Staubli VAL3: RemoteAxisCtrl.pjx

--- RemoteAxisCtrl.pjx ---
Parameters version=s7.3.1 stackSize=5000 millimeterUnit=true
Program file=Comunicacion.pgx
Program file=JOGG_PC.pgx
Program file=init.pgx
Program file=set_sign.pgx
Program file=start.pgx
Program file=stop.pgx
Data file=RemoteAxisCtrl.dtx

--- RemoteAxisCtrl.dtx ---
bool bABSOLUTE = true
bool bBLOQ_CTRL
bool bBusy
bool bError
bool bHoming = true
bool bNewMove
bool bSTOP = true
bool bSync = true
dio Electrovalvule[2]
  [0] = {link=valve1}
  [1] = {link=valve2}
dio dBIO_salidas[4]
  [0] = {link=BasicIO-1\%Q0}
  [1] = {link=BasicIO-1\%Q1}
  [2] = {link=BasicIO-1\%Q2}
  [3] = {link=BasicIO-1\%Q3}
jointRx home = {j2=60, j3=60, j5=60}
jointRx jActualPos = {j2=60, j3=60, j5=60}
jointRx jError = {j1=0.1, j2=0.1, j3=0.1, j4=0.1, j5=0.1, j6=0.1}
jointRx jdestino = {j2=60, j3=60, j5=60}
jointRx origen
mdesc mNomSpeed = {blend=off}
mdesc mSpeed = {vel=10, blend=off}
num action
num axis_v[6]
  [5] = 1
num d_min = 0.5
num error_code
num g_data[82]
  [0] = 156
  [1] = 124
  [2] = 66
  [3] = 89
  [4] = 39
  [5] = 121
  [6] = 244
  [7] = 77
  [12] = 66
  [18] = 128
  [20] = 20
  [21] = 10
  [42] = 100
num g_message_send[82]
  [0] = 156
  [1] = 124
  [2] = 66
  [3] = 89
  [4] = 39
  [5] = 121
  [6] = 244
  [7] = 77
  [12] = 66
  [16] = 32
  [20] = 20
  [21] = 10
  [22] = 250
  [23] = 202
  [26] = 208
  [27] = 7
  [30] = 64
  [31] = 31
  [34] = 80
  [35] = 70
  [42] = 80
  [43] = 70
  [48] = 1
  [49] = 1
  [51] = 1
num id = -1
num id_actual = -2
num joint_v[6]
num mode_mov
num move_inc = 1
num nBytes
num n_status = 1
num speed = 10
num working_mode
pointRx pActualPos = {x=519.615242, y=20, z=-80, rx=-180, rz=-180, shoulder=lefty, elbow=epositive, wrist=wpositive, fatherId=world[0]}
pointRx pPunto = {fatherId=world[0]}
pointRx pdestino = {x=539.615242, y=40, z=-60, rx=-160, ry=20, rz=-160, shoulder=lefty, elbow=epositive, wrist=wpositive, fatherId=world[0]}
sio sSockPC = {link=Socket\RemoteCTRL}
tool tGripper = {fatherId=flange[0], ioLink=valve1}

--- start.pgx ---
program start()
begin
  call init()

  while (bBLOQ_CTRL==false)
    call Comunicacion()
    call JOGG_PC()
    delay(0)
  endWhile

end

--- Comunicacion.pgx ---
program Comunicacion()
  local num i
  local num aux
begin
  //while salir==false
  //communication with the PC
  //Waiting a message from the PC
  nBytes=sioGet(sSockPC,g_data)
  if (nBytes>0)
    //A message was received
    //Reading Identification message (8 bytes). It'll be used in the answer.
    for i=0 to 7
      g_message_send[i]=g_data[i]
    endFor
    //Reserved bytes 8, 9, 10, 11
    //ACTION BYTE 12
    action=g_data[12]
    g_message_send[12]=action
    //Bytes 13, 14 (input reserved). Output -> Status*********************
    //Byte 15 (output error code)******************************
    switch (action)
      case 13
        //NULL ACTION
        //do not do anything.
      break
      case 16
        //READ DATA
        //Update the return data
        //ID message already done
        //Reserved 8, 9, 10, 11
        //ACTION done
        //Status
        g_message_send[13]=n_status
        g_message_send[14]=0
        //Error code
        g_message_send[15]=error_code
        //working mode
        g_message_send[16]=working_mode
        //electrovalvule
        g_message_send[17]=dioGet(Electrovalvule)
        //digital output
        g_message_send[18]=dioGet(dBIO_salidas)
        //DO reserved
        g_message_send[19]=0
        //move inc
        g_message_send[20]=move_inc
        //speed
        g_message_send[21]=speed
        //Actual pos axis
        pActualPos=here(tGripper,world)
        jActualPos=herej()
        call set_sign()
        if (mode_mov==1 or mode_mov==2)
          pActualPos=here(tGripper,world)
          for i=0 to 3
            g_message_send[22+i]=(bAnd(round(abs(pActualPos.trsf.x)*100),power(2,8*(i+1))-power(2,8*i)))/(power(2,8*i))
            g_message_send[26+i]=(bAnd(round(abs(pActualPos.trsf.y)*100),power(2,8*(i+1))-power(2,8*i)))/(power(2,8*i))
            g_message_send[30+i]=(bAnd(round(abs(pActualPos.trsf.z)*100),power(2,8*(i+1))-power(2,8*i)))/(power(2,8*i))
            g_message_send[34+i]=(bAnd(round(abs(pActualPos.trsf.rx)*100),power(2,8*(i+1))-power(2,8*i)))/(power(2,8*i))
            g_message_send[38+i]=(bAnd(round(abs(pActualPos.trsf.ry)*100),power(2,8*(i+1))-power(2,8*i)))/(power(2,8*i))
            g_message_send[42+i]=(bAnd(round(abs(pActualPos.trsf.rz)*100),power(2,8*(i+1))-power(2,8*i)))/(power(2,8*i))
          endFor

          //Actual pos joint
        elseIf (mode_mov==3 or mode_mov==4)
          jActualPos=herej()
          for i=0 to 3
            g_message_send[52+i]=(bAnd(round(abs(jActualPos.j1)*100),power(2,8*(i+1))-power(2,8*i)))/(power(2,8*i))
            g_message_send[56+i]=(bAnd(round(abs(jActualPos.j2)*100),power(2,8*(i+1))-power(2,8*i)))/(power(2,8*i))
            g_message_send[60+i]=(bAnd(round(abs(jActualPos.j3)*100),power(2,8*(i+1))-power(2,8*i)))/(power(2,8*i))
            g_message_send[64+i]=(bAnd(round(abs(jActualPos.j4)*100),power(2,8*(i+1))-power(2,8*i)))/(power(2,8*i))
            g_message_send[68+i]=(bAnd(round(abs(jActualPos.j5)*100),power(2,8*(i+1))-power(2,8*i)))/(power(2,8*i))
            g_message_send[72+i]=(bAnd(round(abs(jActualPos.j6)*100),power(2,8*(i+1))-power(2,8*i)))/(power(2,8*i))
          endFor
        endIf

        //************************************************************************TEMPORAL FALTA SENTIDO EN JOINT Y WORLD ************************************
      break
      case 17
        //WRITE DATA
        //check enable/disable robot motion. stop variable, byte 18
        if (bAnd(g_data[18],1)==1 and bSTOP==true)
          bSTOP=false
          putln("Enabled robot movement")
        elseIf (bAnd(g_data[18],128)==128 and bSTOP==false)
          bSTOP=true
          putln("Erased queue. bSTOP was set up by user.")
        elseIf (bAnd(g_data[18],128)!=128 and bAnd(g_data[18],1)!=1)
          error_code=1
          put("Erased queue. Error at bSTOP input ")
          resetMotion()
        endIf

        //check flag absolute or relative movement. bit 0 (1) byte 19
        if (bABSOLUTE==false and bAnd(g_data[19],1)==1)
          if (bBusy==false)
            bABSOLUTE=true
            putln("Configuration, ABSOLUTE SYSTEM established.")
          else
            error_code=5
            put("Impossible to change system reference. Sys is busy...")
          endIf
        elseIf (bABSOLUTE==true and bAnd(g_data[19],1)==0)
          if (bBusy==false)
            putln("Configuration, RELATIVE SYSTEM established.")
            bABSOLUTE=false
          else
            error_code=5
            put("Impossible to change system reference. Sys is busy...")
          endIf
        elseIf ((bABSOLUTE==true and bAnd(g_data[19],1)==1) or (bABSOLUTE==false and bAnd(g_data[19],1)==0))
          //do not change anything
        else
          //Case not considered
          putln("Case not defined.")
          error_code=13
        endIf

        //check movement config. Bits 2 and 3 ( 4 + 8)
        working_mode=g_data[19]
        if (bAnd(g_data[19],12)==0 and mode_mov!=1)
          //mode 1: axis single
          putln("Mode axis single")
          if (mode_mov==3 or mode_mov==4)
            //change from joint simple/multiple to axis simple
            pdestino=jointToPoint(tGripper,world,jdestino)
          endIf
          mode_mov=1
        elseIf (bAnd(g_data[19],12)==4 and mode_mov!=2)
          //mode 2: axis multiple
          putln("Mode axis multiple")
          if (mode_mov==3 or mode_mov==4)
            //change from joint simple/multiple to axis simple
            pdestino=jointToPoint(tGripper,world,jdestino)
          endIf
          mode_mov=2
        elseIf (bAnd(g_data[19],12)==8 and mode_mov!=3)
          //mode 3: joint single
          if (mode_mov==1 or mode_mov==2)
            //change from joint simple/multiple to axis simple
            pointToJoint(tGripper,jActualPos,pdestino,jdestino)
          endIf
          putln("Mode joint single")
          mode_mov=3
        elseIf (bAnd(g_data[19],12)==12 and mode_mov!=4)
          putln("Mode joint multiple")
          //mode 4: joint multiple
          mode_mov=4
        endIf

        //check flags homing
        if (bAnd(g_data[19],32)==32)
          if (bHoming==false and bBLOQ_CTRL==false and bSTOP==false)
            //go home flag
            put("Erased queue due to homing instruction.")
            resetMotion()
            jdestino=home
            movej(jdestino,tGripper,mNomSpeed)
            //movej(home,tGripper,mNomSpeed)
            bSTOP=true
            bHoming=true
            bBusy=true
            n_status=32
          else
            error_code=5
            putln("Couldn't make homing")
          endIf
        else
          //flag gohome is not up
        endIf

        //Erase queue instruction
        if (bAnd(g_data[19],64)==64)
          //erase queue
          put("Queue erased due to instruction flag.")
          resetMotion()
        endIf

        //Sync or async movement. Can only be changed when robot is not busy.
        if (bSync==false)
          if (bAnd(g_data[19],128)==128 and bBusy==false)
            bSync=true
          elseIf (bAnd(g_data[19],128)==128)
            error_code=5
            putln("Couldn't change movement config")
          endIf
        else
          if (bAnd(g_data[19],128)==0 and bBusy==false)
            bSync=false
          elseIf (bAnd(g_data[19],128)==0)
            error_code=5
            putln("Couldn't change movement config")
          endIf
        endIf

        //inc
        move_inc=g_data[20]
        //speed
        speed=g_data[21]
        //read movement config. Divide per 100 to recover mm. And add sign.
        for i=0 to 5
          if (g_data[46+i]==0)
            aux=1
          else
            aux=-1
          endIf
          axis_v[i]=aux*(g_data[22+4*i]+power(2,8)*g_data[22+4*i+1]+power(2,16)*g_data[22+4*i+2]+power(2,24)*g_data[22+4*i+3])/100
        endFor
        for i=0 to 5
          if (g_data[76+i]==0)
            aux=1
          else
            aux=-1
          endIf
          joint_v[i]=aux*(g_data[52+4*i]+power(2,8)*g_data[52+4*i+1]+power(2,16)*g_data[52+4*i+2]+power(2,24)*g_data[52+4*i+3])/100
        endFor
      break

      case 18
        //SET OUTPUT
        if (g_data[15]>128)
          //set off electrovalvule
          Electrovalvule[g_data[15]-128-1]=false
        elseIf (g_data[15]>0)
          //set on electrovalvule
          Electrovalvule[g_data[15]-1]=true
        endIf
        if (g_data[16]>128)
          //set off digital output
          dBIO_salidas[g_data[16]-128-1]=false
        elseIf (g_data[16]>0)
          dBIO_salidas[g_data[16]-1]=true
        endIf
      break

      case 19
        //START MOVE
        //check axis or joint. Check sync or async.
        //add new move
        if (bAnd(g_data[19],16)==16 and bNewMove==false and bSTOP==false and bBLOQ_CTRL==false and bHoming==false and mode_mov>=1 and mode_mov<=4)
          //start flag
          if (bSync==true and bBusy==false)
            putln("New move input made")
            bNewMove=true
            bBusy=true
          elseIf (bSync==false)
            bNewMove=true
          else
            error_code=4
            putln("Couldn't make a new move")
            //n_status
          endIf
        else
          putln("Impossible to add new move")
          error_code=3
        endIf
      break

      case 66
        //END CONTROL
        bBLOQ_CTRL=true
      break

      default
      break

    endSwitch
    g_message_send[15]=error_code
    sioSet(sSockPC,g_message_send)
  else
    //Message reception failure
    putln("Error, communication")
    resetMotion()
    bBLOQ_CTRL=true
    call stop()
  endIf
  //endWhile
end

--- init.pgx ---
program init()
  local num i
begin
  cls()
  bBLOQ_CTRL=false
  bSTOP=true
  //absolute == false, means relative movement configuration.
  bABSOLUTE=true
  bSync=true
  bBusy=false
  bNewMove=false
  bHoming=true
  nBytes=0
  id=-1
  id_actual=-2
  move_inc=1
  error_code=0
  mode_mov=0
  n_status=1
  speed=10
  mSpeed.vel=speed
  action=0
  d_min=0.5
  //taskCreate "comun", 80, Comunicacion()
  i=movej(origen,flange,mNomSpeed)
  putln("Movimiento a origen 0 ")
  put(i)
  waitEndMove()
  i=movej(home,flange,mNomSpeed)
  putln("Movimiento a home ")
  put(i)
  waitEndMove()
  bHoming=false
  jActualPos=herej()
  pActualPos=here(tGripper,world)
  jdestino=herej()
  pdestino=here(tGripper,world)
  jError={0.1,0.1,0.1,0.1,0.1,0.1}
  //taskCreate "movimiento", 100, JOGG_PC()
  for i=0 to 81
    g_data[i]=0
    g_message_send[i]=0
  endFor
  for i=0 to 5
    axis_v[i]=0
    joint_v[i]=0
  endFor
end

--- JOGG_PC.pgx ---
program JOGG_PC()
  local num l_aux
begin
  if (bBLOQ_CTRL==false and bSTOP==false and bHoming==false and bNewMove)
    //Absolute or relative movement
    if (bABSOLUTE)
      //ABSOLUTE MOVEMENT. ONLY MULTIPLE JOINT AND AXIS
      if (mode_mov==4)
        //Joint multiple
        jdestino.j1=joint_v[0]
        jdestino.j2=joint_v[1]
        jdestino.j3=joint_v[2]
        jdestino.j4=joint_v[3]
        jdestino.j5=joint_v[4]
        jdestino.j6=joint_v[5]
        id=movej(jdestino,tGripper,mSpeed)
        bNewMove=false
        n_status=14
      elseIf (mode_mov==2)
        //Axis multiple
        //pdestino.config = config(jdestino)
        pdestino.trsf.x=axis_v[0]
        pdestino.trsf.y=axis_v[1]
        pdestino.trsf.z=axis_v[2]
        pdestino.trsf.rx=axis_v[3]
        pdestino.trsf.ry=axis_v[4]
        pdestino.trsf.rz=axis_v[5]
        movej(pdestino,tGripper,mSpeed)
        //movel(pdestino,tGripper,mSpeed)
        bNewMove=false
        n_status=12
      else
        //Can not make a single axis/joint movement with ABSOLUTE reference configuration
        putln("Error type movement sel.")
        bBusy=false
        n_status=33
      endIf
    else
      //RELATIVE MOVEMENT
      if (mode_mov==1 or mode_mov==2)
        //axis single/multiple
        if (mode_mov==1)
          l_aux=move_inc
        else
          l_aux=1
        endIf
        if (bSync==true)
          pActualPos=here(tGripper,world)
        else
          pActualPos=pdestino
        endIf
        pdestino.trsf.x=pActualPos.trsf.x+l_aux*axis_v[0]
        pdestino.trsf.y=pActualPos.trsf.y+l_aux*axis_v[1]
        pdestino.trsf.z=pActualPos.trsf.z+l_aux*axis_v[2]
        pdestino.trsf.rx=pActualPos.trsf.rx+l_aux*axis_v[3]
        pdestino.trsf.ry=pActualPos.trsf.ry+l_aux*axis_v[4]
        pdestino.trsf.rz=pActualPos.trsf.rz+l_aux*axis_v[5]
        //id=movel(pdestino,tGripper,mSpeed)
        id=movej(pdestino,tGripper,mSpeed)
        bNewMove=false
        put("Moving from:  ")
        put(pActualPos.trsf.x)
        put(" to: ")
        put(pdestino.trsf.x)
        putln("OK, movej called. ID: ")
        //putln("OK, movel called. ID: ")
        put(id)
        n_status=12
      elseIf (mode_mov==3 or mode_mov==4)
        //multiple/single joint
        if (mode_mov==3)
          l_aux=move_inc
        else
          l_aux=1
        endIf
        jActualPos=herej()
        jdestino.j1=jdestino.j1+l_aux*joint_v[0]
        jdestino.j2=jdestino.j2+l_aux*joint_v[1]
        jdestino.j3=jdestino.j3+l_aux*joint_v[2]
        jdestino.j4=jdestino.j4+l_aux*joint_v[3]
        jdestino.j5=jdestino.j5+l_aux*joint_v[4]
        jdestino.j6=jdestino.j6+l_aux*joint_v[5]
        id=movej(jdestino,tGripper,mSpeed)
        putln("OK, movej called. ID: ")
        //putln("OK, movel called. ID: ")
        put(id)
        bNewMove=false
        n_status=14
      else
        //Wrong mode_mov
        putln("Wrong mode movement")
        bBusy=false
        n_status=111
      endIf
    endIf
  elseIf (bHoming)
    jActualPos=herej()
    if (isEmpty()==true and abs(home-jActualPos)<jError)
      bSTOP=false
      bHoming=false
      bBusy=false
      putln("Homing ended...")
      n_status=0
    endIf
  elseIf (bNewMove)
    bBusy=false
    putln("Tried new move but was impossible...")
    error_code=5
  elseIf (bBusy==true and bSync==true and bBLOQ_CTRL==false and bSTOP==false and bHoming==false)
    if (n_status==12 and isEmpty()==true and distance(pdestino.trsf,pActualPos.trsf)<1)
      bBusy=false
      putln("Movement ended (12)...")
      n_status=0
    elseIf (n_status==14 and isEmpty()==true and abs(jdestino-jActualPos)<jError)
      bBusy=false
      putln("Movement ended (14)...")
      n_status=0
    endIf
  elseIf (bBLOQ_CTRL==false and bSTOP==false and bBusy==false)
    //Complete this part of the code..................................................
    pActualPos=here(tGripper,world)
    jActualPos=herej()
    id_actual=roundDown(getMoveId())
    if (isEmpty()==true and isSettled()==true and id_actual>=id)
      if ((mode_mov<=2 and distance(pdestino.trsf,pActualPos.trsf)<1) or (mode_mov>2 and abs(jdestino-jActualPos)<jError))
        n_status=0
        put("Valor de id actual:  ")
        put(id_actual)
        putln("..>=.. ")
        put("Valor de getMoveId al cancelar: ")
        put(id)
      endIf
    endIf
  elseIf (bSTOP==true or bBLOQ_CTRL==true)
    resetMotion()
  else
    put("Undefined error")
    error_code=13
  endIf
end

--- set_sign.pgx ---
program set_sign()
begin
  if (pActualPos.trsf.x>=0)
    g_message_send[46]=0
  else
    g_message_send[46]=1
  endIf
  if (pActualPos.trsf.y>=0)
    g_message_send[47]=0
  else
    g_message_send[47]=1
  endIf
  if (pActualPos.trsf.z>=0)
    g_message_send[48]=0
  else
    g_message_send[48]=1
  endIf
  if (pActualPos.trsf.rx>=0)
    g_message_send[49]=0
  else
    g_message_send[49]=1
  endIf
  if (pActualPos.trsf.ry>=0)
    g_message_send[50]=0
  else
    g_message_send[50]=1
  endIf
  if (pActualPos.trsf.rz>=0)
    g_message_send[51]=0
  else
    g_message_send[51]=1
  endIf


  if (jActualPos.j1>=0)
    g_message_send[76]=0
  else
    g_message_send[76]=1
  endIf
  if (jActualPos.j2>=0)
    g_message_send[77]=0
  else
    g_message_send[77]=1
  endIf
  if (jActualPos.j3>=0)
    g_message_send[78]=0
  else
    g_message_send[78]=1
  endIf
  if (jActualPos.j4>=0)
    g_message_send[79]=0
  else
    g_message_send[79]=1
  endIf
  if (jActualPos.j5>=0)
    g_message_send[80]=0
  else
    g_message_send[80]=1
  endIf
  if (jActualPos.j6>=0)
    g_message_send[81]=0
  else
    g_message_send[81]=1
  endIf





end

--- stop.pgx ---
program stop()
begin
  stopMove()
  resetMotion()
  clearBuffer(sSockPC)
end
